Staubli VAL3: stopAreaTest.pgx

public program stopAreaTest(bool& bResult_[])
begin
  // test result of area test state machine
  // the state nAreaTestState must be 40
  if nAreaTestState!=40 and nAreaTestState!=0
    call status:raise(AREA_TEST_FAIL,"")
  endIf
  bResult_=nAreaTestState==40 or nAreaTestState==0
end
